FUNCTION_BLOCK SS0_ifb_magzine (* Basic FB with empty ECC *)
  (* Standard: 61499-2 *)
  (* Version 1.0, 2025-04-16, DEVIASH *)
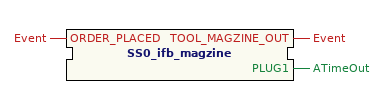
  EVENT_INPUT
    ORDER_PLACED;
  END_EVENT
  EVENT_OUTPUT
    TOOL_MAGZINE_OUT;
  END_EVENT
  PLUGS
    PLUG1 : ATimeOut;
  END_PLUGS
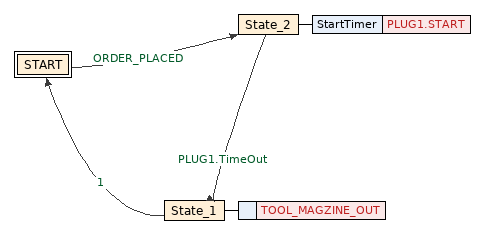
  EC_STATES
    START; (* Initial State *)
    State_2 : StartTimer -> PLUG1.START;
    State_1 : -> TOOL_MAGZINE_OUT;
  END_STATES
  EC_TRANSITIONS
    START TO State_2 := ORDER_PLACED;
    State_2 TO State_1 := PLUG1.TimeOut;
    State_1 TO START := 1;
  END_TRANSITIONS
  ALGORITHM StartTimer IN ST:
PLUG1.DT := T#12s;
  END_ALGORITHM
END_FUNCTION_BLOCK
